LIN {X 0,Y 75.955,Z 312.798,A -85,B 0,C 180,E1 -27969.999,E2 -27969.999} C_VEL
LIN {X 0,Y 72.056,Z 313.683,A -85,B 0,C 180,E1 -27975.335,E2 -27975.335} C_VEL
LIN {X 0,Y 70.252,Z 314.024,A -85,B 0,C 180,E1 -27979.881,E2 -27979.881} C_VEL
LIN {X 0,Y 69.991,Z 314.033,A -85,B 0,C 180,E1 -27981.483,E2 -27981.483} C_VEL
LIN {X 0,Y 69.758,Z 313.788,A -85,B 0,C 180,E1 -27989.996,E2 -27989.996} C_VEL
LIN {X 0,Y 70.22,Z 313.122,A -85,B 0,C 180,E1 -27995.74,E2 -27995.74} C_VEL
LIN {X 0,Y 71.125,Z 312.075,A -85,B 0,C 180,E1 -28001.393,E2 -28001.393} C_VEL
LIN {X 0,Y 72.573,Z 310.585,A -85,B 0,C 180,E1 -28006.884,E2 -28006.884} C_VEL
LIN {X 0,Y 75.758,Z 307.579,A -85,B 0,C 180,E1 -28014.668,E2 -28014.668} C_VEL
LIN {X 0,Y 80.142,Z 303.529,A -85,B 0,C 180,E1 -28021.74,E2 -28021.74} C_VEL
LIN {X 0,Y 86.545,Z 297.313,A -85,B 0,C 180,E1 -28028.995,E2 -28028.995} C_VEL
LIN {X 0,Y 92.996,Z 290.542,A -85,B 0,C 180,E1 -28034.343,E2 -28034.343} C_VEL
LIN {X 0,Y 98.789,Z 283.636,A -85,B 0,C 180,E1 -28038.321,E2 -28038.321} C_VEL
LIN {X 0,Y 101.219,Z 280.484,A -85,B 0,C 180,E1 -28039.788,E2 -28039.788} C_VEL
LIN {X 0,Y 102.858,Z 276.343,A -85,B 0,C 180,E1 -28042.553,E2 -28042.553} C_VEL
LIN {X 0,Y 103.486,Z 273.641,A -85,B 0,C 180,E1 -28044.572,E2 -28044.572} C_VEL
LIN {X 0,Y 103.73,Z 270.638,A -85,B 0,C 180,E1 -28047.177,E2 -28047.177} C_VEL
LIN {X 0,Y 103.119,Z 265.886,A -85,B 0,C 180,E1 -28052.362,E2 -28052.362} C_VEL
LIN {X 0,Y 102.624,Z 263.228,A -85,B 0,C 180,E1 -28055.738,E2 -28055.738} C_VEL
LIN {X 0,Y 101.676,Z 259.362,A -85,B 0,C 180,E1 -28061.877,E2 -28061.877} C_VEL
LIN {X 0,Y 100.935,Z 256.73,A -85,B 0,C 180,E1 -28067.942,E2 -28067.942} C_VEL
LIN {X 0,Y 100.648,Z 254.765,A -85,B 0,C 180,E1 -28075.995,E2 -28075.995} C_VEL
LIN {X 0,Y 100.96,Z 254.248,A -85,B 0,C 180,E1 -28079.999,E2 -28079.999} C_VEL
LIN {X 0,Y 101.079,Z 256.427,A -85,B 0,C 180,E1 -28087.993,E2 -28087.993} C_VEL
LIN {X 0,Y 101.672,Z 257.847,A -85,B 0,C 180,E1 -28091.968,E2 -28091.968} C_VEL
LIN {X 0,Y 102.317,Z 259.954,A -85,B 0,C 180,E1 -28095.946,E2 -28095.946} C_VEL
LIN {X 0,Y 102.785,Z 262.952,A -85,B 0,C 180,E1 -28099.991,E2 -28099.991} C_VEL
LIN {X 0,Y 103.035,Z 267.977,A -85,B 0,C 180,E1 -28105.157,E2 -28105.157} C_VEL
LIN {X 0,Y 103.023,Z 272.964,A -85,B 0,C 180,E1 -28109.641,E2 -28109.641} C_VEL
LIN {X 0,Y 102.775,Z 275.854,A -85,B 0,C 180,E1 -28112.002,E2 -28112.002} C_VEL
LIN {X 0,Y 100.768,Z 280.852,A -85,B 0,C 180,E1 -28114.976,E2 -28114.976} C_VEL
LIN {X 0,Y 97.27,Z 287.517,A -85,B 0,C 180,E1 -28119.049,E2 -28119.049} C_VEL
LIN {X 0,Y 90.366,Z 295.686,A -85,B 0,C 180,E1 -28124.004,E2 -28124.004} C_VEL
LIN {X 0,Y 85.188,Z 301.246,A -85,B 0,C 180,E1 -28128.708,E2 -28128.708} C_VEL
LIN {X 0,Y 79.619,Z 306.676,A -85,B 0,C 180,E1 -28134.994,E2 -28134.994} C_VEL
LIN {X 0,Y 75.07,Z 310.919,A -85,B 0,C 180,E1 -28142.096,E2 -28142.096} C_VEL
LIN {X 0,Y 72.862,Z 313.178,A -85,B 0,C 180,E1 -28147.311,E2 -28147.311} C_VEL
LIN {X 0,Y 71.207,Z 314.96,A -85,B 0,C 180,E1 -28152.782,E2 -28152.782} C_VEL
LIN {X 0,Y 70.138,Z 316.312,A -85,B 0,C 180,E1 -28158.444,E2 -28158.444} C_VEL
LIN {X 0,Y 69.618,Z 317.268,A -85,B 0,C 180,E1 -28164.21,E2 -28164.21} C_VEL
LIN {X 0,Y 69.673,Z 317.834,A -85,B 0,C 180,E1 -28170.004,E2 -28170.004} C_VEL
LIN {X 0,Y 69.621,Z 317.95,A -85,B 0,C 180,E1 -28175.797,E2 -28175.797} C_VEL
LIN {X 0,Y 70.144,Z 317.665,A -85,B 0,C 180,E1 -28181.563,E2 -28181.563} C_VEL
LIN {X 0,Y 72.933,Z 315.942,A -85,B 0,C 180,E1 -28192.674,E2 -28192.674} C_VEL
LIN {X 0,Y 75.178,Z 314.45,A -85,B 0,C 180,E1 -28197.869,E2 -28197.869} C_VEL
LIN {X 0,Y 79.764,Z 311.427,A -85,B 0,C 180,E1 -28204.941,E2 -28204.941} C_VEL
LIN {X 0,Y 85.398,Z 307.36,A -85,B 0,C 180,E1 -28211.177,E2 -28211.177} C_VEL
LIN {X 0,Y 92.891,Z 301.121,A -85,B 0,C 180,E1 -28217.532,E2 -28217.532} C_VEL
LIN {X 0,Y 100.186,Z 294.343,A -85,B 0,C 180,E1 -28222.108,E2 -28222.108} C_VEL
LIN {X 0,Y 102.526,Z 291.722,A -85,B 0,C 180,E1 -28223.652,E2 -28223.652} C_VEL
LIN {X 0,Y 106.564,Z 285.03,A -85,B 0,C 180,E1 -28228.157,E2 -28228.157} C_VEL
LIN {X 0,Y 107.391,Z 281.213,A -85,B 0,C 180,E1 -28231.636,E2 -28231.636} C_VEL
LIN {X 0,Y 107.939,Z 276.036,A -85,B 0,C 180,E1 -28237.005,E2 -28237.005} C_VEL
LIN {X 0,Y 108.074,Z 272.768,A -85,B 0,C 180,E1 -28241.026,E2 -28241.026} C_VEL
LIN {X 0,Y 108.135,Z 270.019,A -85,B 0,C 180,E1 -28244.932,E2 -28244.932} C_VEL
LIN {X 0,Y 108.02,Z 268.068,A -85,B 0,C 180,E1 -28248.745,E2 -28248.745} C_VEL
LIN {X 0,Y 107.866,Z 266.689,A -85,B 0,C 180,E1 -28252.513,E2 -28252.513} C_VEL
LIN {X 0,Y 107.979,Z 265.237,A -85,B 0,C 180,E1 -28260.001,E2 -28260.001} C_VEL
LIN {X 0,Y 107.676,Z 266.885,A -85,B 0,C 180,E1 -28267.765,E2 -28267.765} C_VEL
LIN {X 0,Y 107.883,Z 268.439,A -85,B 0,C 180,E1 -28272.273,E2 -28272.273} C_VEL
LIN {X 0,Y 108.215,Z 270.725,A -85,B 0,C 180,E1 -28276.994,E2 -28276.994} C_VEL
LIN {X 0,Y 108.545,Z 274.554,A -85,B 0,C 180,E1 -28282.861,E2 -28282.861} C_VEL
LIN {X 0,Y 108.197,Z 278.26,A -85,B 0,C 180,E1 -28287.046,E2 -28287.046} C_VEL
LIN {X 0,Y 107.345,Z 282.888,A -85,B 0,C 180,E1 -28291.667,E2 -28291.667} C_VEL
LIN {X 0,Y 106.008,Z 285.83,A -85,B 0,C 180,E1 -28294.035,E2 -28294.035} C_VEL
LIN {X 0,Y 104.982,Z 287.233,A -85,B 0,C 180,E1 -28294.909,E2 -28294.909} C_VEL
LIN {X 0,Y 97.412,Z 294.692,A -85,B 0,C 180,E1 -28299.143,E2 -28299.143} C_VEL
LIN {X 0,Y 89.39,Z 301.569,A -85,B 0,C 180,E1 -28304.96,E2 -28304.96} C_VEL
LIN {X 0,Y 83.435,Z 306.095,A -85,B 0,C 180,E1 -28310.82,E2 -28310.82} C_VEL
LIN {X 0,Y 77.622,Z 309.911,A -85,B 0,C 180,E1 -28318.44,E2 -28318.44} C_VEL
LIN {X 0,Y 73.212,Z 312.551,A -85,B 0,C 180,E1 -28327.417,E2 -28327.417} C_VEL
LIN {X 0,Y 71.531,Z 313.461,A -85,B 0,C 180,E1 -28332.855,E2 -28332.855} C_VEL
LIN {X 0,Y 69.991,Z 314.033,A -85,B 0,C 180,E1 -28341.483,E2 -28341.483} C_VEL
LIN {X 0,Y 69.438,Z 314.073,A -85,B 0,C 180,E1 -28344.684,E2 -28344.684} C_VEL
LIN {X 0,Y 68.018,Z 313.906,A -85,B 0,C 180,E1 -28349.481,E2 -28349.481} C_VEL
LIN {X 0,Y 64.974,Z 312.491,A -85,B 0,C 180,E1 -28361.198,E2 -28361.198} C_VEL
LIN {X 0,Y 65.187,Z 311.42,A -85,B 0,C 180,E1 -28366.375,E2 -28366.375} C_VEL
LIN {X 0,Y 65.618,Z 310.972,A -85,B 0,C 180,E1 -28368.043,E2 -28368.043} C_VEL
LIN {X 0,Y 69.372,Z 307.82,A -85,B 0,C 180,E1 -28377.116,E2 -28377.116} C_VEL
LIN {X 0,Y 74.216,Z 303.782,A -85,B 0,C 180,E1 -28384.616,E2 -28384.616} C_VEL
LIN {X 0,Y 81.161,Z 297.581,A -85,B 0,C 180,E1 -28392.143,E2 -28392.143} C_VEL
LIN {X 0,Y 88.063,Z 290.826,A -85,B 0,C 180,E1 -28397.57,E2 -28397.57} C_VEL
LIN {X 0,Y 95.523,Z 282.413,A -85,B 0,C 180,E1 -28402.262,E2 -28402.262} C_VEL
LIN {X 0,Y 96.961,Z 279.827,A -85,B 0,C 180,E1 -28403.959,E2 -28403.959} C_VEL
LIN {X 0,Y 97.919,Z 277.001,A -85,B 0,C 180,E1 -28406.203,E2 -28406.203} C_VEL
LIN {X 0,Y 98.319,Z 274.084,A -85,B 0,C 180,E1 -28409.056,E2 -28409.056} C_VEL
LIN {X 0,Y 98.185,Z 271.419,A -85,B 0,C 180,E1 -28412.301,E2 -28412.301} C_VEL
LIN {X 0,Y 97.853,Z 268.184,A -85,B 0,C 180,E1 -28416.731,E2 -28416.731} C_VEL
LIN {X 0,Y 97.258,Z 264.548,A -85,B 0,C 180,E1 -28423.198,E2 -28423.198} C_VEL
LIN {X 0,Y 96.959,Z 262.844,A -85,B 0,C 180,E1 -28427.439,E2 -28427.439} C_VEL
LIN {X 0,Y 96.783,Z 260.823,A -85,B 0,C 180,E1 -28435.835,E2 -28435.835} C_VEL
LIN {X 0,Y 97.132,Z 260.307,A -85,B 0,C 180,E1 -28439.999,E2 -28439.999} C_VEL
LIN {X 0,Y 97.154,Z 262.517,A -85,B 0,C 180,E1 -28448.318,E2 -28448.318} C_VEL
LIN {X 0,Y 97.649,Z 264.033,A -85,B 0,C 180,E1 -28452.468,E2 -28452.468} C_VEL
LIN {X 0,Y 97.966,Z 266.405,A -85,B 0,C 180,E1 -28456.675,E2 -28456.675} C_VEL
LIN {X 0,Y 98.12,Z 267.867,A -85,B 0,C 180,E1 -28458.802,E2 -28458.802} C_VEL
LIN {X 0,Y 97.911,Z 272.888,A -85,B 0,C 180,E1 -28464.374,E2 -28464.374} C_VEL
LIN {X 0,Y 97.466,Z 277.636,A -85,B 0,C 180,E1 -28468.998,E2 -28468.998} C_VEL
LIN {X 0,Y 96.932,Z 279.503,A -85,B 0,C 180,E1 -28470.499,E2 -28470.499} C_VEL
LIN {X 0,Y 93.687,Z 285.648,A -85,B 0,C 180,E1 -28474.405,E2 -28474.405} C_VEL
LIN {X 0,Y 91.691,Z 288.714,A -85,B 0,C 180,E1 -28476.418,E2 -28476.418} C_VEL
LIN {X 0,Y 84.392,Z 296.628,A -85,B 0,C 180,E1 -28481.462,E2 -28481.462} C_VEL
LIN {X 0,Y 77.841,Z 302.947,A -85,B 0,C 180,E1 -28487.387,E2 -28487.387} C_VEL
LIN {X 0,Y 72.098,Z 307.974,A -85,B 0,C 180,E1 -28494.214,E2 -28494.214} C_VEL
LIN {X 0,Y 67.496,Z 311.866,A -85,B 0,C 180,E1 -28502.066,E2 -28502.066} C_VEL
LIN {X 0,Y 64.441,Z 314.737,A -85,B 0,C 180,E1 -28510.908,E2 -28510.908} C_VEL
LIN {X 0,Y 63.173,Z 316.095,A -85,B 0,C 180,E1 -28517.149,E2 -28517.149} C_VEL
LIN {X 0,Y 62.553,Z 317.057,A -85,B 0,C 180,E1 -28523.554,E2 -28523.554} C_VEL
LIN {X 0,Y 62.564,Z 317.628,A -85,B 0,C 180,E1 -28530.004,E2 -28530.004} C_VEL
LIN {X 0,Y 62.556,Z 317.754,A -85,B 0,C 180,E1 -28536.455,E2 -28536.455} C_VEL
LIN {X 0,Y 64.469,Z 316.812,A -85,B 0,C 180,E1 -28549.092,E2 -28549.092} C_VEL
LIN {X 0,Y 66.394,Z 315.762,A -85,B 0,C 180,E1 -28555.053,E2 -28555.053} C_VEL
LIN {X 0,Y 68.957,Z 314.281,A -85,B 0,C 180,E1 -28560.639,E2 -28560.639} C_VEL
LIN {X 0,Y 74.036,Z 311.27,A -85,B 0,C 180,E1 -28568.101,E2 -28568.101} C_VEL
LIN {X 0,Y 80.179,Z 307.215,A -85,B 0,C 180,E1 -28574.526,E2 -28574.526} C_VEL
LIN {X 0,Y 88.233,Z 300.99,A -85,B 0,C 180,E1 -28580.951,E2 -28580.951} C_VEL
LIN {X 0,Y 95.975,Z 294.228,A -85,B 0,C 180,E1 -28585.467,E2 -28585.467} C_VEL
LIN {X 0,Y 97.202,Z 292.973,A -85,B 0,C 180,E1 -28586.251,E2 -28586.251} C_VEL
LIN {X 0,Y 100.572,Z 288.15,A -85,B 0,C 180,E1 -28589.722,E2 -28589.722} C_VEL
LIN {X 0,Y 101.23,Z 286.76,A -85,B 0,C 180,E1 -28590.924,E2 -28590.924} C_VEL
LIN {X 0,Y 102.278,Z 282.398,A -85,B 0,C 180,E1 -28595.652,E2 -28595.652} C_VEL
LIN {X 0,Y 102.847,Z 278.852,A -85,B 0,C 180,E1 -28600.022,E2 -28600.022} C_VEL
LIN {X 0,Y 103.165,Z 276.019,A -85,B 0,C 180,E1 -28604.188,E2 -28604.188} C_VEL
LIN {X 0,Y 103.363,Z 273.814,A -85,B 0,C 180,E1 -28608.231,E2 -28608.231} C_VEL
LIN {X 0,Y 103.361,Z 272.372,A -85,B 0,C 180,E1 -28612.185,E2 -28612.185} C_VEL
LIN {X 0,Y 103.556,Z 270.864,A -85,B 0,C 180,E1 -28620.001,E2 -28620.001} C_VEL
LIN {X 0,Y 103.125,Z 272.419,A -85,B 0,C 180,E1 -28627.835,E2 -28627.835} C_VEL
LIN {X 0,Y 103.164,Z 273.663,A -85,B 0,C 180,E1 -28631.794,E2 -28631.794} C_VEL
LIN {X 0,Y 103.269,Z 276.393,A -85,B 0,C 180,E1 -28637.683,E2 -28637.683} C_VEL
LIN {X 0,Y 103.251,Z 279.001,A -85,B 0,C 180,E1 -28641.986,E2 -28641.986} C_VEL
LIN {X 0,Y 102.452,Z 283.012,A -85,B 0,C 180,E1 -28646.905,E2 -28646.905} C_VEL
LIN {X 0,Y 101.988,Z 284.706,A -85,B 0,C 180,E1 -28648.842,E2 -28648.842} C_VEL
LIN {X 0,Y 100.629,Z 287.643,A -85,B 0,C 180,E1 -28651.611,E2 -28651.611} C_VEL
LIN {X 0,Y 95.729,Z 292.503,A -85,B 0,C 180,E1 -28654.319,E2 -28654.319} C_VEL
LIN {X 0,Y 89.284,Z 297.98,A -85,B 0,C 180,E1 -28658.08,E2 -28658.08} C_VEL
LIN {X 0,Y 82.425,Z 303.193,A -85,B 0,C 180,E1 -28663.262,E2 -28663.262} C_VEL
LIN {X 0,Y 76.073,Z 307.488,A -85,B 0,C 180,E1 -28669.706,E2 -28669.706} C_VEL
LIN {X 0,Y 72.408,Z 309.696,A -85,B 0,C 180,E1 -28674.381,E2 -28674.381} C_VEL
LIN {X 0,Y 69.213,Z 311.423,A -85,B 0,C 180,E1 -28679.487,E2 -28679.487} C_VEL
LIN {X 0,Y 64.762,Z 313.646,A -85,B 0,C 180,E1 -28690.997,E2 -28690.997} C_VEL
LIN {X 0,Y 62.938,Z 314.236,A -85,B 0,C 180,E1 -28700.978,E2 -28700.978} C_VEL
LIN {X 0,Y 62.679,Z 313.994,A -85,B 0,C 180,E1 -28709.996,E2 -28709.996} C_VEL
LIN {X 0,Y 63.18,Z 313.334,A -85,B 0,C 180,E1 -28716.382,E2 -28716.382} C_VEL
LIN {X 0,Y 64.189,Z 312.294,A -85,B 0,C 180,E1 -28722.644,E2 -28722.644} C_VEL
LIN {X 0,Y 65.618,Z 310.972,A -85,B 0,C 180,E1 -28728.043,E2 -28728.043} C_VEL
LIN {X 0,Y 66.735,Z 309.623,A -85,B 0,C 180,E1 -28732.928,E2 -28732.928} C_VEL
LIN {X 0,Y 67.72,Z 306.86,A -85,B 0,C 180,E1 -28741.014,E2 -28741.014} C_VEL
LIN {X 0,Y 69.774,Z 303.403,A -85,B 0,C 180,E1 -28748.598,E2 -28748.598} C_VEL
LIN {X 0,Y 72.402,Z 300.889,A -85,B 0,C 180,E1 -28752.383,E2 -28752.383} C_VEL
LIN {X 0,Y 79.684,Z 294.661,A -85,B 0,C 180,E1 -28758.553,E2 -28758.553} C_VEL
LIN {X 0,Y 87.32,Z 287.157,A -85,B 0,C 180,E1 -28763.585,E2 -28763.585} C_VEL
LIN {X 0,Y 90.886,Z 283.208,A -85,B 0,C 180,E1 -28765.616,E2 -28765.616} C_VEL
LIN {X 0,Y 91.978,Z 281.164,A -85,B 0,C 180,E1 -28767.182,E2 -28767.182} C_VEL
LIN {X 0,Y 92.61,Z 279.392,A -85,B 0,C 180,E1 -28768.899,E2 -28768.899} C_VEL
LIN {X 0,Y 92.87,Z 277.921,A -85,B 0,C 180,E1 -28770.534,E2 -28770.534} C_VEL
LIN {X 0,Y 92.877,Z 274.63,A -85,B 0,C 180,E1 -28775.22,E2 -28775.22} C_VEL
LIN {X 0,Y 92.789,Z 271.95,A -85,B 0,C 180,E1 -28779.698,E2 -28779.698} C_VEL
LIN {X 0,Y 92.742,Z 270.542,A -85,B 0,C 180,E1 -28782.354,E2 -28782.354} C_VEL
LIN {X 0,Y 92.552,Z 268.768,A -85,B 0,C 180,E1 -28786.831,E2 -28786.831} C_VEL
LIN {X 0,Y 92.461,Z 267.552,A -85,B 0,C 180,E1 -28791.255,E2 -28791.255} C_VEL
LIN {X 0,Y 92.585,Z 266.672,A -85,B 0,C 180,E1 -28795.646,E2 -28795.646} C_VEL
LIN {X 0,Y 92.963,Z 266.166,A -85,B 0,C 180,E1 -28799.999,E2 -28799.999} C_VEL
LIN {X 0,Y 93.061,Z 269.154,A -85,B 0,C 180,E1 -28810.995,E2 -28810.995} C_VEL
LIN {X 0,Y 93.254,Z 271.189,A -85,B 0,C 180,E1 -28815.293,E2 -28815.293} C_VEL
LIN {X 0,Y 93.259,Z 272.612,A -85,B 0,C 180,E1 -28817.543,E2 -28817.543} C_VEL
LIN {X 0,Y 92.739,Z 276.431,A -85,B 0,C 180,E1 -28822.266,E2 -28822.266} C_VEL
LIN {X 0,Y 91.913,Z 281.062,A -85,B 0,C 180,E1 -28827.308,E2 -28827.308} C_VEL
LIN {X 0,Y 90.911,Z 283.114,A -85,B 0,C 180,E1 -28828.871,E2 -28828.871} C_VEL
LIN {X 0,Y 87.528,Z 288.405,A -85,B 0,C 180,E1 -28832.545,E2 -28832.545} C_VEL
LIN {X 0,Y 82.366,Z 293.881,A -85,B 0,C 180,E1 -28835.857,E2 -28835.857} C_VEL
LIN {X 0,Y 75.004,Z 300.708,A -85,B 0,C 180,E1 -28841.453,E2 -28841.453} C_VEL
LIN {X 0,Y 68.403,Z 306.168,A -85,B 0,C 180,E1 -28848.109,E2 -28848.109} C_VEL
LIN {X 0,Y 62.842,Z 310.439,A -85,B 0,C 180,E1 -28856.009,E2 -28856.009} C_VEL
LIN {X 0,Y 59.914,Z 312.707,A -85,B 0,C 180,E1 -28862.024,E2 -28862.024} C_VEL
LIN {X 0,Y 57.732,Z 314.513,A -85,B 0,C 180,E1 -28868.587,E2 -28868.587} C_VEL
LIN {X 0,Y 56.261,Z 315.878,A -85,B 0,C 180,E1 -28875.538,E2 -28875.538} C_VEL
LIN {X 0,Y 55.511,Z 316.846,A -85,B 0,C 180,E1 -28882.732,E2 -28882.732} C_VEL
LIN {X 0,Y 55.475,Z 317.423,A -85,B 0,C 180,E1 -28890.005,E2 -28890.005} C_VEL
LIN {X 0,Y 55.514,Z 317.56,A -85,B 0,C 180,E1 -28897.278,E2 -28897.278} C_VEL
LIN {X 0,Y 57.779,Z 316.627,A -85,B 0,C 180,E1 -28911.405,E2 -28911.405} C_VEL
LIN {X 0,Y 59.996,Z 315.582,A -85,B 0,C 180,E1 -28917.944,E2 -28917.944} C_VEL
LIN {X 0,Y 62.934,Z 314.113,A -85,B 0,C 180,E1 -28923.945,E2 -28923.945} C_VEL
LIN {X 0,Y 68.56,Z 311.112,A -85,B 0,C 180,E1 -28931.784,E2 -28931.784} C_VEL
LIN {X 0,Y 76.758,Z 306.048,A -85,B 0,C 180,E1 -28939.59,E2 -28939.59} C_VEL
LIN {X 0,Y 85.25,Z 299.849,A -85,B 0,C 180,E1 -28945.527,E2 -28945.527} C_VEL
LIN {X 0,Y 92.072,Z 294.113,A -85,B 0,C 180,E1 -28949.173,E2 -28949.173} C_VEL
LIN {X 0,Y 95.249,Z 290.122,A -85,B 0,C 180,E1 -28952.302,E2 -28952.302} C_VEL
LIN {X 0,Y 96.261,Z 287.575,A -85,B 0,C 180,E1 -28955.178,E2 -28955.178} C_VEL
LIN {X 0,Y 97.295,Z 283.977,A -85,B 0,C 180,E1 -28959.888,E2 -28959.888} C_VEL
LIN {X 0,Y 98.086,Z 280.469,A -85,B 0,C 180,E1 -28965.477,E2 -28965.477} C_VEL
LIN {X 0,Y 98.338,Z 279.317,A -85,B 0,C 180,E1 -28967.62,E2 -28967.62} C_VEL
LIN {X 0,Y 98.478,Z 277.804,A -85,B 0,C 180,E1 -28971.795,E2 -28971.795} C_VEL
LIN {X 0,Y 98.61,Z 276.782,A -85,B 0,C 180,E1 -28976.167,E2 -28976.167} C_VEL
LIN {X 0,Y 98.836,Z 276.237,A -85,B 0,C 180,E1 -28980.001,E2 -28980.001} C_VEL
LIN {X 0,Y 98.214,Z 277.777,A -85,B 0,C 180,E1 -28988.229,E2 -28988.229} C_VEL
LIN {X 0,Y 98.119,Z 279.1,A -85,B 0,C 180,E1 -28992.41,E2 -28992.41} C_VEL
LIN {X 0,Y 98.04,Z 280.861,A -85,B 0,C 180,E1 -28996.664,E2 -28996.664} C_VEL
LIN {X 0,Y 97.763,Z 283.271,A -85,B 0,C 180,E1 -29001.067,E2 -29001.067} C_VEL
LIN {X 0,Y 96.663,Z 286.791,A -85,B 0,C 180,E1 -29005.865,E2 -29005.865} C_VEL
LIN {X 0,Y 95.743,Z 288.803,A -85,B 0,C 180,E1 -29008.256,E2 -29008.256} C_VEL
LIN {X 0,Y 94.676,Z 290.141,A -85,B 0,C 180,E1 -29009.283,E2 -29009.283} C_VEL
LIN {X 0,Y 86.405,Z 297.105,A -85,B 0,C 180,E1 -29013.518,E2 -29013.518} C_VEL
LIN {X 0,Y 78.409,Z 302.867,A -85,B 0,C 180,E1 -29018.863,E2 -29018.863} C_VEL
LIN {X 0,Y 70.778,Z 307.643,A -85,B 0,C 180,E1 -29025.965,E2 -29025.965} C_VEL
LIN {X 0,Y 66.758,Z 309.858,A -85,B 0,C 180,E1 -29030.826,E2 -29030.826} C_VEL
LIN {X 0,Y 63.172,Z 311.596,A -85,B 0,C 180,E1 -29036.2,E2 -29036.2} C_VEL
LIN {X 0,Y 58.085,Z 313.83,A -85,B 0,C 180,E1 -29048.713,E2 -29048.713} C_VEL
LIN {X 0,Y 56.522,Z 314.367,A -85,B 0,C 180,E1 -29055.596,E2 -29055.596} C_VEL
LIN {X 0,Y 55.692,Z 314.479,A -85,B 0,C 180,E1 -29062.746,E2 -29062.746} C_VEL
LIN {X 0,Y 55.591,Z 314.2,A -85,B 0,C 180,E1 -29069.995,E2 -29069.995} C_VEL
LIN {X 0,Y 56.136,Z 313.545,A -85,B 0,C 180,E1 -29077.187,E2 -29077.187} C_VEL
LIN {X 0,Y 57.283,Z 312.513,A -85,B 0,C 180,E1 -29084.198,E2 -29084.198} C_VEL
LIN {X 0,Y 59.154,Z 311.042,A -85,B 0,C 180,E1 -29090.874,E2 -29090.874} C_VEL
LIN {X 0,Y 63.146,Z 308.061,A -85,B 0,C 180,E1 -29100.048,E2 -29100.048} C_VEL
LIN {X 0,Y 68.486,Z 304.037,A -85,B 0,C 180,E1 -29107.996,E2 -29107.996} C_VEL
LIN {X 0,Y 72.402,Z 300.889,A -85,B 0,C 180,E1 -29112.383,E2 -29112.383} C_VEL
LIN {X 0,Y 76.26,Z 297.24,A -85,B 0,C 180,E1 -29116.848,E2 -29116.848} C_VEL
LIN {X 0,Y 79.485,Z 293.298,A -85,B 0,C 180,E1 -29121.286,E2 -29121.286} C_VEL
LIN {X 0,Y 82.645,Z 289.036,A -85,B 0,C 180,E1 -29125.484,E2 -29125.484} C_VEL
LIN {X 0,Y 86.2,Z 284.363,A -85,B 0,C 180,E1 -29129.147,E2 -29129.147} C_VEL
LIN {X 0,Y 87.106,Z 282.499,A -85,B 0,C 180,E1 -29131.045,E2 -29131.045} C_VEL
LIN {X 0,Y 87.439,Z 280.718,A -85,B 0,C 180,E1 -29133.564,E2 -29133.564} C_VEL
LIN {X 0,Y 87.75,Z 277.549,A -85,B 0,C 180,E1 -29138.873,E2 -29138.873} C_VEL
LIN {X 0,Y 87.814,Z 275.307,A -85,B 0,C 180,E1 -29143.796,E2 -29143.796} C_VEL
LIN {X 0,Y 87.824,Z 273.171,A -85,B 0,C 180,E1 -29150.789,E2 -29150.789} C_VEL
LIN {X 0,Y 88.071,Z 272.274,A -85,B 0,C 180,E1 -29155.422,E2 -29155.422} C_VEL
LIN {X 0,Y 88.49,Z 271.776,A -85,B 0,C 180,E1 -29159.999,E2 -29159.999} C_VEL
LIN {X 0,Y 88.259,Z 273.997,A -85,B 0,C 180,E1 -29169.163,E2 -29169.163} C_VEL
LIN {X 0,Y 88.35,Z 275.805,A -85,B 0,C 180,E1 -29173.805,E2 -29173.805} C_VEL
LIN {X 0,Y 87.833,Z 278.866,A -85,B 0,C 180,E1 -29178.666,E2 -29178.666} C_VEL
LIN {X 0,Y 86.745,Z 283.013,A -85,B 0,C 180,E1 -29183.896,E2 -29183.896} C_VEL
LIN {X 0,Y 85.9,Z 284.975,A -85,B 0,C 180,E1 -29185.86,E2 -29185.86} C_VEL
LIN {X 0,Y 82.522,Z 289.579,A -85,B 0,C 180,E1 -29189.212,E2 -29189.212} C_VEL
LIN {X 0,Y 74.455,Z 297.113,A -85,B 0,C 180,E1 -29194.136,E2 -29194.136} C_VEL
LIN {X 0,Y 65.596,Z 304.247,A -85,B 0,C 180,E1 -29201.422,E2 -29201.422} C_VEL
LIN {X 0,Y 59.015,Z 308.914,A -85,B 0,C 180,E1 -29209.091,E2 -29209.091} C_VEL
LIN {X 0,Y 53.706,Z 312.471,A -85,B 0,C 180,E1 -29218.445,E2 -29218.445} C_VEL
LIN {X 0,Y 51.145,Z 314.289,A -85,B 0,C 180,E1 -29225.662,E2 -29225.662} C_VEL
LIN {X 0,Y 49.382,Z 315.66,A -85,B 0,C 180,E1 -29233.47,E2 -29233.47} C_VEL
LIN {X 0,Y 48.471,Z 316.634,A -85,B 0,C 180,E1 -29241.669,E2 -29241.669} C_VEL
LIN {X 0,Y 48.372,Z 317.217,A -85,B 0,C 180,E1 -29250.006,E2 -29250.006} C_VEL
LIN {X 0,Y 48.474,Z 317.364,A -85,B 0,C 180,E1 -29258.341,E2 -29258.341} C_VEL
LIN {X 0,Y 51.195,Z 316.441,A -85,B 0,C 180,E1 -29274.324,E2 -29274.324} C_VEL
LIN {X 0,Y 53.789,Z 315.402,A -85,B 0,C 180,E1 -29281.513,E2 -29281.513} C_VEL
LIN {X 0,Y 57.168,Z 313.946,A -85,B 0,C 180,E1 -29287.931,E2 -29287.931} C_VEL
LIN {X 0,Y 63.409,Z 310.954,A -85,B 0,C 180,E1 -29296.092,E2 -29296.092} C_VEL
LIN {X 0,Y 70.716,Z 306.923,A -85,B 0,C 180,E1 -29302.663,E2 -29302.663} C_VEL
LIN {X 0,Y 80.015,Z 300.73,A -85,B 0,C 180,E1 -29308.912,E2 -29308.912} C_VEL
LIN {X 0,Y 87.183,Z 295.234,A -85,B 0,C 180,E1 -29312.464,E2 -29312.464} C_VEL
LIN {X 0,Y 89.542,Z 292.736,A -85,B 0,C 180,E1 -29314.502,E2 -29314.502} C_VEL
LIN {X 0,Y 90.652,Z 290.58,A -85,B 0,C 180,E1 -29317.194,E2 -29317.194} C_VEL
LIN {X 0,Y 91.984,Z 287.226,A -85,B 0,C 180,E1 -29322.206,E2 -29322.206} C_VEL
LIN {X 0,Y 92.843,Z 284.701,A -85,B 0,C 180,E1 -29326.875,E2 -29326.875} C_VEL
LIN {X 0,Y 93.118,Z 283.788,A -85,B 0,C 180,E1 -29328.855,E2 -29328.855} C_VEL
LIN {X 0,Y 93.256,Z 282.972,A -85,B 0,C 180,E1 -29331.332,E2 -29331.332} C_VEL
LIN {X 0,Y 93.512,Z 281.908,A -85,B 0,C 180,E1 -29335.691,E2 -29335.691} C_VEL
LIN {X 0,Y 93.805,Z 281.306,A -85,B 0,C 180,E1 -29340.001,E2 -29340.001} C_VEL
LIN {X 0,Y 93,Z 282.694,A -85,B 0,C 180,E1 -29347.781,E2 -29347.781} C_VEL
LIN {X 0,Y 92.747,Z 284.25,A -85,B 0,C 180,E1 -29353.141,E2 -29353.141} C_VEL
LIN {X 0,Y 92.41,Z 286.092,A -85,B 0,C 180,E1 -29357.712,E2 -29357.712} C_VEL
LIN {X 0,Y 91.953,Z 287.681,A -85,B 0,C 180,E1 -29360.67,E2 -29360.67} C_VEL
LIN {X 0,Y 91.02,Z 289.796,A -85,B 0,C 180,E1 -29363.913,E2 -29363.913} C_VEL
LIN {X 0,Y 89.925,Z 291.501,A -85,B 0,C 180,E1 -29366.005,E2 -29366.005} C_VEL
LIN {X 0,Y 81.277,Z 298.237,A -85,B 0,C 180,E1 -29370.153,E2 -29370.153} C_VEL
LIN {X 0,Y 73.656,Z 303.312,A -85,B 0,C 180,E1 -29374.926,E2 -29374.926} C_VEL
LIN {X 0,Y 65.821,Z 307.799,A -85,B 0,C 180,E1 -29381.631,E2 -29381.631} C_VEL
LIN {X 0,Y 61.389,Z 310.02,A -85,B 0,C 180,E1 -29386.613,E2 -29386.613} C_VEL
LIN {X 0,Y 57.384,Z 311.77,A -85,B 0,C 180,E1 -29392.237,E2 -29392.237} C_VEL
LIN {X 0,Y 51.503,Z 314.014,A -85,B 0,C 180,E1 -29405.831,E2 -29405.831} C_VEL
LIN {X 0,Y 49.671,Z 314.558,A -85,B 0,C 180,E1 -29413.557,E2 -29413.557} C_VEL
LIN {X 0,Y 48.648,Z 314.679,A -85,B 0,C 180,E1 -29421.689,E2 -29421.689} C_VEL
LIN {X 0,Y 48.492,Z 314.406,A -85,B 0,C 180,E1 -29429.994,E2 -29429.994} C_VEL
LIN {X 0,Y 49.127,Z 313.756,A -85,B 0,C 180,E1 -29438.219,E2 -29438.219} C_VEL
LIN {X 0,Y 50.447,Z 312.73,A -85,B 0,C 180,E1 -29446.172,E2 -29446.172} C_VEL
LIN {X 0,Y 52.578,Z 311.271,A -85,B 0,C 180,E1 -29453.634,E2 -29453.634} C_VEL
LIN {X 0,Y 57.129,Z 308.301,A -85,B 0,C 180,E1 -29463.605,E2 -29463.605} C_VEL
LIN {X 0,Y 63.044,Z 304.29,A -85,B 0,C 180,E1 -29471.97,E2 -29471.97} C_VEL
LIN {X 0,Y 71.299,Z 298.116,A -85,B 0,C 180,E1 -29479.801,E2 -29479.801} C_VEL
LIN {X 0,Y 79.192,Z 291.392,A -85,B 0,C 180,E1 -29485.163,E2 -29485.163} C_VEL
LIN {X 0,Y 85.705,Z 284.987,A -85,B 0,C 180,E1 -29488.722,E2 -29488.722} C_VEL
LIN {X 0,Y 86.2,Z 284.363,A -85,B 0,C 180,E1 -29489.147,E2 -29489.147} C_VEL
LIN {X 0,Y 87.266,Z 282.59,A -85,B 0,C 180,E1 -29490.781,E2 -29490.781} C_VEL
LIN {X 0,Y 87.507,Z 280.959,A -85,B 0,C 180,E1 -29493.33,E2 -29493.33} C_VEL
LIN {X 0,Y 86.651,Z 279.713,A -85,B 0,C 180,E1 -29497.106,E2 -29497.106} C_VEL
LIN {X 0,Y 83.938,Z 279.115,A -85,B 0,C 180,E1 -29504.281,E2 -29504.281} C_VEL
LIN {X 0,Y 82.865,Z 278.5,A -85,B 0,C 180,E1 -29510.426,E2 -29510.426} C_VEL
LIN {X 0,Y 83.193,Z 277.606,A -85,B 0,C 180,E1 -29515.153,E2 -29515.153} C_VEL
LIN {X 0,Y 83.685,Z 277.124,A -85,B 0,C 180,E1 -29519.999,E2 -29519.999} C_VEL
LIN {X 0,Y 83.308,Z 278.122,A -85,B 0,C 180,E1 -29524.838,E2 -29524.838} C_VEL
LIN {X 0,Y 83.241,Z 279.417,A -85,B 0,C 180,E1 -29529.72,E2 -29529.72} C_VEL
LIN {X 0,Y 83.209,Z 280.297,A -85,B 0,C 180,E1 -29532.189,E2 -29532.189} C_VEL
LIN {X 0,Y 82.649,Z 282.527,A -85,B 0,C 180,E1 -29536.415,E2 -29536.415} C_VEL
LIN {X 0,Y 81.229,Z 286.311,A -85,B 0,C 180,E1 -29541.803,E2 -29541.803} C_VEL
LIN {X 0,Y 80.299,Z 287.756,A -85,B 0,C 180,E1 -29543.239,E2 -29543.239} C_VEL
LIN {X 0,Y 77.823,Z 290.654,A -85,B 0,C 180,E1 -29545.451,E2 -29545.451} C_VEL
LIN {X 0,Y 68.894,Z 298.276,A -85,B 0,C 180,E1 -29550.473,E2 -29550.473} C_VEL
LIN {X 0,Y 61.12,Z 303.987,A -85,B 0,C 180,E1 -29556.412,E2 -29556.412} C_VEL
LIN {X 0,Y 53.83,Z 308.667,A -85,B 0,C 180,E1 -29564.115,E2 -29564.115} C_VEL
LIN {X 0,Y 47.768,Z 312.236,A -85,B 0,C 180,E1 -29573.958,E2 -29573.958} C_VEL
LIN {X 0,Y 44.738,Z 314.065,A -85,B 0,C 180,E1 -29581.892,E2 -29581.892} C_VEL
LIN {X 0,Y 42.599,Z 315.442,A -85,B 0,C 180,E1 -29590.742,E2 -29590.742} C_VEL
LIN {X 0,Y 41.444,Z 316.422,A -85,B 0,C 180,E1 -29600.244,E2 -29600.244} C_VEL
LIN {X 0,Y 41.285,Z 317.012,A -85,B 0,C 180,E1 -29610.007,E2 -29610.007} C_VEL
LIN {X 0,Y 41.448,Z 317.169,A -85,B 0,C 180,E1 -29619.768,E2 -29619.768} C_VEL
LIN {X 0,Y 44.788,Z 316.256,A -85,B 0,C 180,E1 -29638.088,E2 -29638.088} C_VEL
LIN {X 0,Y 47.847,Z 315.222,A -85,B 0,C 180,E1 -29645.987,E2 -29645.987} C_VEL
LIN {X 0,Y 51.743,Z 313.778,A -85,B 0,C 180,E1 -29652.778,E2 -29652.778} C_VEL
LIN {X 0,Y 58.682,Z 310.795,A -85,B 0,C 180,E1 -29661.122,E2 -29661.122} C_VEL
LIN {X 0,Y 66.623,Z 306.776,A -85,B 0,C 180,E1 -29667.556,E2 -29667.556} C_VEL
LIN {X 0,Y 76.585,Z 300.601,A -85,B 0,C 180,E1 -29673.474,E2 -29673.474} C_VEL
LIN {X 0,Y 82.606,Z 296.306,A -85,B 0,C 180,E1 -29676.147,E2 -29676.147} C_VEL
LIN {X 0,Y 83.924,Z 295.112,A -85,B 0,C 180,E1 -29677.096,E2 -29677.096} C_VEL
LIN {X 0,Y 84.67,Z 294.136,A -85,B 0,C 180,E1 -29678.296,E2 -29678.296} C_VEL
LIN {X 0,Y 86.307,Z 291.069,A -85,B 0,C 180,E1 -29683.442,E2 -29683.442} C_VEL
LIN {X 0,Y 86.93,Z 289.778,A -85,B 0,C 180,E1 -29685.964,E2 -29685.964} C_VEL
LIN {X 0,Y 87.756,Z 287.847,A -85,B 0,C 180,E1 -29690.784,E2 -29690.784} C_VEL
LIN {X 0,Y 88.12,Z 286.723,A -85,B 0,C 180,E1 -29695.427,E2 -29695.427} C_VEL
LIN {X 0,Y 88.482,Z 286.085,A -85,B 0,C 180,E1 -29700.001,E2 -29700.001} C_VEL
LIN {X 0,Y 87.557,Z 287.367,A -85,B 0,C 180,E1 -29707.65,E2 -29707.65} C_VEL
LIN {X 0,Y 87.496,Z 287.687,A -85,B 0,C 180,E1 -29709.246,E2 -29709.246} C_VEL
LIN {X 0,Y 86.741,Z 289.995,A -85,B 0,C 180,E1 -29716.473,E2 -29716.473} C_VEL
LIN {X 0,Y 85.717,Z 292.138,A -85,B 0,C 180,E1 -29720.828,E2 -29720.828} C_VEL
LIN {X 0,Y 83.994,Z 294.057,A -85,B 0,C 180,E1 -29723.017,E2 -29723.017} C_VEL
LIN {X 0,Y 74.998,Z 300.316,A -85,B 0,C 180,E1 -29727.098,E2 -29727.098} C_VEL
LIN {X 0,Y 66.573,Z 305.284,A -85,B 0,C 180,E1 -29732.376,E2 -29732.376} C_VEL
LIN {X 0,Y 58.828,Z 309.124,A -85,B 0,C 180,E1 -29739.053,E2 -29739.053} C_VEL
LIN {X 0,Y 51.931,Z 311.943,A -85,B 0,C 180,E1 -29747.413,E2 -29747.413} C_VEL
LIN {X 0,Y 45.1,Z 314.199,A -85,B 0,C 180,E1 -29762.124,E2 -29762.124} C_VEL
LIN {X 0,Y 42.888,Z 314.749,A -85,B 0,C 180,E1 -29770.863,E2 -29770.863} C_VEL
LIN {X 0,Y 41.641,Z 314.88,A -85,B 0,C 180,E1 -29780.277,E2 -29780.277} C_VEL
LIN {X 0,Y 41.41,Z 314.611,A -85,B 0,C 180,E1 -29789.993,E2 -29789.993} C_VEL
LIN {X 0,Y 42.128,Z 313.967,A -85,B 0,C 180,E1 -29799.596,E2 -29799.596} C_VEL
LIN {X 0,Y 43.674,Z 312.947,A -85,B 0,C 180,E1 -29808.766,E2 -29808.766} C_VEL
LIN {X 0,Y 46.166,Z 311.5,A -85,B 0,C 180,E1 -29817.165,E2 -29817.165} C_VEL
LIN {X 0,Y 51.367,Z 308.542,A -85,B 0,C 180,E1 -29827.992,E2 -29827.992} C_VEL
LIN {X 0,Y 57.967,Z 304.543,A -85,B 0,C 180,E1 -29836.662,E2 -29836.662} C_VEL
LIN {X 0,Y 66.948,Z 298.383,A -85,B 0,C 180,E1 -29844.434,E2 -29844.434} C_VEL
LIN {X 0,Y 75.369,Z 291.674,A -85,B 0,C 180,E1 -29849.588,E2 -29849.588} C_VEL
LIN {X 0,Y 81.203,Z 286.331,A -85,B 0,C 180,E1 -29852.469,E2 -29852.469} C_VEL
LIN {X 0,Y 81.837,Z 284.827,A -85,B 0,C 180,E1 -29854.57,E2 -29854.57} C_VEL
LIN {X 0,Y 82.447,Z 281.923,A -85,B 0,C 180,E1 -29860.063,E2 -29860.063} C_VEL
LIN {X 0,Y 82.744,Z 279.889,A -85,B 0,C 180,E1 -29865.236,E2 -29865.236} C_VEL
LIN {X 0,Y 82.865,Z 278.5,A -85,B 0,C 180,E1 -29870.426,E2 -29870.426} C_VEL
LIN {X 0,Y 82.439,Z 278.552,A -85,B 0,C 180,E1 -29873.114,E2 -29873.114} C_VEL
LIN {X 0,Y 81.018,Z 279.765,A -85,B 0,C 180,E1 -29876.595,E2 -29876.595} C_VEL
LIN {X 0,Y 78.387,Z 282.606,A -85,B 0,C 180,E1 -29882.918,E2 -29882.918} C_VEL
LIN {X 0,Y 78.126,Z 283.13,A -85,B 0,C 180,E1 -29884.879,E2 -29884.879} C_VEL
LIN {X 0,Y 77.93,Z 284.554,A -85,B 0,C 180,E1 -29890.39,E2 -29890.39} C_VEL
LIN {X 0,Y 77.598,Z 285.641,A -85,B 0,C 180,E1 -29893.085,E2 -29893.085} C_VEL
LIN {X 0,Y 76.28,Z 288.417,A -85,B 0,C 180,E1 -29897.894,E2 -29897.894} C_VEL
LIN {X 0,Y 74.854,Z 290.341,A -85,B 0,C 180,E1 -29900.156,E2 -29900.156} C_VEL
LIN {X 0,Y 73.484,Z 291.725,A -85,B 0,C 180,E1 -29901.194,E2 -29901.194} C_VEL
LIN {X 0,Y 65.856,Z 297.778,A -85,B 0,C 180,E1 -29904.918,E2 -29904.918} C_VEL
LIN {X 0,Y 57.179,Z 303.727,A -85,B 0,C 180,E1 -29910.656,E2 -29910.656} C_VEL
LIN {X 0,Y 49.134,Z 308.419,A -85,B 0,C 180,E1 -29918.135,E2 -29918.135} C_VEL
LIN {X 0,Y 42.203,Z 312,A -85,B 0,C 180,E1 -29928.244,E2 -29928.244} C_VEL
LIN {X 0,Y 38.596,Z 313.842,A -85,B 0,C 180,E1 -29936.9,E2 -29936.9} C_VEL
LIN {X 0,Y 35.957,Z 315.224,A -85,B 0,C 180,E1 -29946.999,E2 -29946.999} C_VEL
LIN {X 0,Y 34.465,Z 316.211,A -85,B 0,C 180,E1 -29958.243,E2 -29958.243} C_VEL
LIN {X 0,Y 34.174,Z 316.805,A -85,B 0,C 180,E1 -29970.008,E2 -29970.008} C_VEL
LIN {X 0,Y 34.47,Z 316.973,A -85,B 0,C 180,E1 -29981.772,E2 -29981.772} C_VEL
LIN {X 0,Y 38.644,Z 316.071,A -85,B 0,C 180,E1 -30003.071,E2 -30003.071} C_VEL
LIN {X 0,Y 42.28,Z 315.043,A -85,B 0,C 180,E1 -30011.68,E2 -30011.68} C_VEL
LIN {X 0,Y 46.776,Z 313.609,A -85,B 0,C 180,E1 -30018.702,E2 -30018.702} C_VEL
LIN {X 0,Y 54.488,Z 310.635,A -85,B 0,C 180,E1 -30026.972,E2 -30026.972} C_VEL
LIN {X 0,Y 63.069,Z 306.627,A -85,B 0,C 180,E1 -30033.06,E2 -30033.06} C_VEL
LIN {X 0,Y 73.677,Z 300.472,A -85,B 0,C 180,E1 -30038.44,E2 -30038.44} C_VEL
LIN {X 0,Y 78.402,Z 297.304,A -85,B 0,C 180,E1 -30040.257,E2 -30040.257} C_VEL
LIN {X 0,Y 79.48,Z 296.137,A -85,B 0,C 180,E1 -30041.975,E2 -30041.975} C_VEL
LIN {X 0,Y 80.987,Z 293.868,A -85,B 0,C 180,E1 -30046.551,E2 -30046.551} C_VEL
LIN {X 0,Y 81.741,Z 292.558,A -85,B 0,C 180,E1 -30050.099,E2 -30050.099} C_VEL
LIN {X 0,Y 82.435,Z 291.265,A -85,B 0,C 180,E1 -30055.11,E2 -30055.11} C_VEL
LIN {X 0,Y 82.899,Z 290.572,A -85,B 0,C 180,E1 -30060.001,E2 -30060.001} C_VEL
LIN {X 0,Y 81.822,Z 291.718,A -85,B 0,C 180,E1 -30067.333,E2 -30067.333} C_VEL
LIN {X 0,Y 81.594,Z 292.216,A -85,B 0,C 180,E1 -30069.921,E2 -30069.921} C_VEL
LIN {X 0,Y 80.966,Z 293.648,A -85,B 0,C 180,E1 -30075.095,E2 -30075.095} C_VEL
LIN {X 0,Y 79.809,Z 295.298,A -85,B 0,C 180,E1 -30078.801,E2 -30078.801} C_VEL
LIN {X 0,Y 72.028,Z 300.451,A -85,B 0,C 180,E1 -30082.036,E2 -30082.036} C_VEL
LIN {X 0,Y 63.034,Z 305.434,A -85,B 0,C 180,E1 -30086.878,E2 -30086.878} C_VEL
LIN {X 0,Y 54.616,Z 309.286,A -85,B 0,C 180,E1 -30093.233,E2 -30093.233} C_VEL
LIN {X 0,Y 46.932,Z 312.116,A -85,B 0,C 180,E1 -30101.515,E2 -30101.515} C_VEL
LIN {X 0,Y 38.954,Z 314.383,A -85,B 0,C 180,E1 -30117.226,E2 -30117.226} C_VEL
LIN {X 0,Y 36.246,Z 314.938,A -85,B 0,C 180,E1 -30127.177,E2 -30127.177} C_VEL
LIN {X 0,Y 34.657,Z 315.081,A -85,B 0,C 180,E1 -30138.293,E2 -30138.293} C_VEL
LIN {X 0,Y 34.311,Z 314.818,A -85,B 0,C 180,E1 -30149.992,E2 -30149.992} C_VEL
LIN {X 0,Y 35.152,Z 314.179,A -85,B 0,C 180,E1 -30161.524,E2 -30161.524} C_VEL
LIN {X 0,Y 37.038,Z 313.164,A -85,B 0,C 180,E1 -30172.293,E2 -30172.293} C_VEL
LIN {X 0,Y 39.996,Z 311.728,A -85,B 0,C 180,E1 -30181.803,E2 -30181.803} C_VEL
LIN {X 0,Y 45.986,Z 308.781,A -85,B 0,C 180,E1 -30193.439,E2 -30193.439} C_VEL
LIN {X 0,Y 53.355,Z 304.794,A -85,B 0,C 180,E1 -30202.202,E2 -30202.202} C_VEL
LIN {X 0,Y 63.093,Z 298.65,A -85,B 0,C 180,E1 -30209.671,E2 -30209.671} C_VEL
LIN {X 0,Y 72.043,Z 291.957,A -85,B 0,C 180,E1 -30214.453,E2 -30214.453} C_VEL
LIN {X 0,Y 75.849,Z 288.712,A -85,B 0,C 180,E1 -30216.167,E2 -30216.167} C_VEL
LIN {X 0,Y 76.3,Z 288.066,A -85,B 0,C 180,E1 -30217.068,E2 -30217.068} C_VEL
LIN {X 0,Y 76.758,Z 286.709,A -85,B 0,C 180,E1 -30219.993,E2 -30219.993} C_VEL
LIN {X 0,Y 77.233,Z 285.093,A -85,B 0,C 180,E1 -30224.156,E2 -30224.156} C_VEL
LIN {X 0,Y 77.656,Z 283.355,A -85,B 0,C 180,E1 -30231.094,E2 -30231.094} C_VEL
LIN {X 0,Y 78.008,Z 282.675,A -85,B 0,C 180,E1 -30234.83,E2 -30234.83} C_VEL
LIN {X 0,Y 78.567,Z 282.17,A -85,B 0,C 180,E1 -30239.999,E2 -30239.999} C_VEL
LIN {X 0,Y 78.126,Z 283.13,A -85,B 0,C 180,E1 -30244.879,E2 -30244.879} C_VEL
LIN {X 0,Y 77.536,Z 284.25,A -85,B 0,C 180,E1 -30247.776,E2 -30247.776} C_VEL
LIN {X 0,Y 76.194,Z 286.037,A -85,B 0,C 180,E1 -30250.409,E2 -30250.409} C_VEL
LIN {X 0,Y 73.557,Z 289.022,A -85,B 0,C 180,E1 -30253.495,E2 -30253.495} C_VEL
LIN {X 0,Y 70.106,Z 292.292,A -85,B 0,C 180,E1 -30256.027,E2 -30256.027} C_VEL
LIN {X 0,Y 68.08,Z 293.907,A -85,B 0,C 180,E1 -30256.984,E2 -30256.984} C_VEL
LIN {X 0,Y 58.053,Z 300.914,A -85,B 0,C 180,E1 -30261.542,E2 -30261.542} C_VEL
LIN {X 0,Y 47.918,Z 306.735,A -85,B 0,C 180,E1 -30268.376,E2 -30268.376} C_VEL
LIN {X 0,Y 39.683,Z 310.691,A -85,B 0,C 180,E1 -30277.176,E2 -30277.176} C_VEL
LIN {X 0,Y 32.846,Z 313.617,A -85,B 0,C 180,E1 -30290.08,E2 -30290.08} C_VEL
LIN {X 0,Y 29.518,Z 315.006,A -85,B 0,C 180,E1 -30301.576,E2 -30301.576} C_VEL
LIN {X 0,Y 27.534,Z 315.999,A -85,B 0,C 180,E1 -30315.223,E2 -30315.223} C_VEL
LIN {X 0,Y 27.066,Z 316.599,A -85,B 0,C 180,E1 -30330.01,E2 -30330.01} C_VEL
LIN {X 0,Y 27.54,Z 316.777,A -85,B 0,C 180,E1 -30344.794,E2 -30344.794} C_VEL
LIN {X 0,Y 32.907,Z 315.887,A -85,B 0,C 180,E1 -30369.853,E2 -30369.853} C_VEL
LIN {X 0,Y 37.254,Z 314.863,A -85,B 0,C 180,E1 -30378.997,E2 -30378.997} C_VEL
LIN {X 0,Y 42.406,Z 313.439,A -85,B 0,C 180,E1 -30385.967,E2 -30385.967} C_VEL
LIN {X 0,Y 50.956,Z 310.475,A -85,B 0,C 180,E1 -30393.704,E2 -30393.704} C_VEL
LIN {X 0,Y 60.17,Z 306.479,A -85,B 0,C 180,E1 -30399.137,E2 -30399.137} C_VEL
LIN {X 0,Y 71.372,Z 300.342,A -85,B 0,C 180,E1 -30403.756,E2 -30403.756} C_VEL
LIN {X 0,Y 73.009,Z 299.331,A -85,B 0,C 180,E1 -30404.284,E2 -30404.284} C_VEL
LIN {X 0,Y 74.737,Z 297.772,A -85,B 0,C 180,E1 -30406.919,E2 -30406.919} C_VEL
LIN {X 0,Y 75.375,Z 296.926,A -85,B 0,C 180,E1 -30409.254,E2 -30409.254} C_VEL
LIN {X 0,Y 76.404,Z 295.517,A -85,B 0,C 180,E1 -30414.723,E2 -30414.723} C_VEL
LIN {X 0,Y 77.053,Z 294.764,A -85,B 0,C 180,E1 -30420.001,E2 -30420.001} C_VEL
LIN {X 0,Y 75.908,Z 295.692,A -85,B 0,C 180,E1 -30426.787,E2 -30426.787} C_VEL
LIN {X 0,Y 75.106,Z 296.934,A -85,B 0,C 180,E1 -30432.891,E2 -30432.891} C_VEL
LIN {X 0,Y 74.387,Z 297.723,A -85,B 0,C 180,E1 -30435.001,E2 -30435.001} C_VEL
LIN {X 0,Y 63.266,Z 304.037,A -85,B 0,C 180,E1 -30439.225,E2 -30439.225} C_VEL
LIN {X 0,Y 54.011,Z 308.266,A -85,B 0,C 180,E1 -30444.374,E2 -30444.374} C_VEL
LIN {X 0,Y 48.146,Z 310.504,A -85,B 0,C 180,E1 -30448.852,E2 -30448.852} C_VEL
LIN {X 0,Y 42.547,Z 312.29,A -85,B 0,C 180,E1 -30454.315,E2 -30454.315} C_VEL
LIN {X 0,Y 33.19,Z 314.568,A -85,B 0,C 180,E1 -30470.554,E2 -30470.554} C_VEL
LIN {X 0,Y 29.83,Z 315.128,A -85,B 0,C 180,E1 -30481.879,E2 -30481.879} C_VEL
LIN {X 0,Y 27.73,Z 315.282,A -85,B 0,C 180,E1 -30495.31,E2 -30495.31} C_VEL
LIN {X 0,Y 27.228,Z 315.023,A -85,B 0,C 180,E1 -30509.99,E2 -30509.99} C_VEL
LIN {X 0,Y 28.251,Z 314.39,A -85,B 0,C 180,E1 -30524.394,E2 -30524.394} C_VEL
LIN {X 0,Y 30.598,Z 313.381,A -85,B 0,C 180,E1 -30537.335,E2 -30537.335} C_VEL
LIN {X 0,Y 34.171,Z 311.957,A -85,B 0,C 180,E1 -30548.085,E2 -30548.085} C_VEL
LIN {X 0,Y 41.132,Z 309.02,A -85,B 0,C 180,E1 -30560.239,E2 -30560.239} C_VEL
LIN {X 0,Y 49.336,Z 305.044,A -85,B 0,C 180,E1 -30568.71,E2 -30568.71} C_VEL
LIN {X 0,Y 59.83,Z 298.917,A -85,B 0,C 180,E1 -30575.535,E2 -30575.535} C_VEL
LIN {X 0,Y 69.082,Z 292.394,A -85,B 0,C 180,E1 -30579.666,E2 -30579.666} C_VEL
LIN {X 0,Y 70.473,Z 291.326,A -85,B 0,C 180,E1 -30580.212,E2 -30580.212} C_VEL
LIN {X 0,Y 71.254,Z 290.121,A -85,B 0,C 180,E1 -30582.787,E2 -30582.787} C_VEL
LIN {X 0,Y 71.945,Z 288.488,A -85,B 0,C 180,E1 -30588.732,E2 -30588.732} C_VEL
LIN {X 0,Y 72.56,Z 287.445,A -85,B 0,C 180,E1 -30594.44,E2 -30594.44} C_VEL
LIN {X 0,Y 73.164,Z 286.944,A -85,B 0,C 180,E1 -30599.999,E2 -30599.999} C_VEL
LIN {X 0,Y 72.662,Z 287.952,A -85,B 0,C 180,E1 -30605.549,E2 -30605.549} C_VEL
LIN {X 0,Y 72.106,Z 289.513,A -85,B 0,C 180,E1 -30611.24,E2 -30611.24} C_VEL
LIN {X 0,Y 71.168,Z 291.009,A -85,B 0,C 180,E1 -30614.289,E2 -30614.289} C_VEL
LIN {X 0,Y 69.593,Z 292.746,A -85,B 0,C 180,E1 -30616.414,E2 -30616.414} C_VEL
LIN {X 0,Y 68.08,Z 293.907,A -85,B 0,C 180,E1 -30616.984,E2 -30616.984} C_VEL
LIN {X 0,Y 63.384,Z 297.2,A -85,B 0,C 180,E1 -30618.273,E2 -30618.273} C_VEL
LIN {X 0,Y 54.785,Z 302.041,A -85,B 0,C 180,E1 -30619.269,E2 -30619.269} C_VEL
LIN {X 0,Y 45.859,Z 306.21,A -85,B 0,C 180,E1 -30620.773,E2 -30620.773} C_VEL
LIN {X 0,Y 40.746,Z 308.397,A -85,B 0,C 180,E1 -30623.462,E2 -30623.462} C_VEL
LIN {X 0,Y 32.955,Z 311.53,A -85,B 0,C 180,E1 -30631.48,E2 -30631.48} C_VEL
LIN {X 0,Y 27.755,Z 313.392,A -85,B 0,C 180,E1 -30640.587,E2 -30640.587} C_VEL
LIN {X 0,Y 23.495,Z 314.788,A -85,B 0,C 180,E1 -30653.273,E2 -30653.273} C_VEL
LIN {X 0,Y 20.741,Z 315.787,A -85,B 0,C 180,E1 -30670.208,E2 -30670.208} C_VEL
LIN {X 0,Y 19.971,Z 316.393,A -85,B 0,C 180,E1 -30690.014,E2 -30690.014} C_VEL
LIN {X 0,Y 20.748,Z 316.58,A -85,B 0,C 180,E1 -30709.812,E2 -30709.812} C_VEL
LIN {X 0,Y 27.807,Z 315.702,A -85,B 0,C 180,E1 -30739.318,E2 -30739.318} C_VEL
LIN {X 0,Y 33.015,Z 314.684,A -85,B 0,C 180,E1 -30748.384,E2 -30748.384} C_VEL
LIN {X 0,Y 38.865,Z 313.269,A -85,B 0,C 180,E1 -30754.716,E2 -30754.716} C_VEL
LIN {X 0,Y 48.227,Z 310.315,A -85,B 0,C 180,E1 -30761.308,E2 -30761.308} C_VEL
LIN {X 0,Y 59.781,Z 305.486,A -85,B 0,C 180,E1 -30766.402,E2 -30766.402} C_VEL
LIN {X 0,Y 67.73,Z 301.372,A -85,B 0,C 180,E1 -30768.892,E2 -30768.892} C_VEL
LIN {X 0,Y 70.024,Z 299.449,A -85,B 0,C 180,E1 -30774.241,E2 -30774.241} C_VEL
LIN {X 0,Y 70.435,Z 299.057,A -85,B 0,C 180,E1 -30776.199,E2 -30776.199} C_VEL
LIN {X 0,Y 70.934,Z 298.597,A -85,B 0,C 180,E1 -30780.001,E2 -30780.001} C_VEL
LIN {X 0,Y 69.507,Z 299.645,A -85,B 0,C 180,E1 -30788.213,E2 -30788.213} C_VEL
LIN {X 0,Y 69.359,Z 299.834,A -85,B 0,C 180,E1 -30789.443,E2 -30789.443} C_VEL
LIN {X 0,Y 67.637,Z 300.905,A -85,B 0,C 180,E1 -30790.934,E2 -30790.934} C_VEL
LIN {X 0,Y 57.994,Z 305.732,A -85,B 0,C 180,E1 -30794.189,E2 -30794.189} C_VEL
LIN {X 0,Y 48.291,Z 309.609,A -85,B 0,C 180,E1 -30798.916,E2 -30798.916} C_VEL
LIN {X 0,Y 38.981,Z 312.463,A -85,B 0,C 180,E1 -30805.642,E2 -30805.642} C_VEL
LIN {X 0,Y 28.046,Z 314.753,A -85,B 0,C 180,E1 -30821.246,E2 -30821.246} C_VEL
LIN {X 0,Y 23.783,Z 315.318,A -85,B 0,C 180,E1 -30833.761,E2 -30833.761} C_VEL
LIN {X 0,Y 20.941,Z 315.482,A -85,B 0,C 180,E1 -30850.378,E2 -30850.378} C_VEL
LIN {X 0,Y 20.119,Z 315.23,A -85,B 0,C 180,E1 -30869.986,E2 -30869.986} C_VEL
LIN {X 0,Y 21.451,Z 314.602,A -85,B 0,C 180,E1 -30889.11,E2 -30889.11} C_VEL
LIN {X 0,Y 24.508,Z 313.598,A -85,B 0,C 180,E1 -30904.98,E2 -30904.98} C_VEL
LIN {X 0,Y 28.914,Z 312.185,A -85,B 0,C 180,E1 -30916.8,E2 -30916.8} C_VEL
LIN {X 0,Y 37.008,Z 309.257,A -85,B 0,C 180,E1 -30928.692,E2 -30928.692} C_VEL
LIN {X 0,Y 46.053,Z 305.295,A -85,B 0,C 180,E1 -30936.272,E2 -30936.272} C_VEL
LIN {X 0,Y 57.252,Z 299.185,A -85,B 0,C 180,E1 -30942.026,E2 -30942.026} C_VEL
LIN {X 0,Y 65.476,Z 293.749,A -85,B 0,C 180,E1 -30944.991,E2 -30944.991} C_VEL
LIN {X 0,Y 65.917,Z 293.055,A -85,B 0,C 180,E1 -30947.686,E2 -30947.686} C_VEL
LIN {X 0,Y 66.771,Z 291.936,A -85,B 0,C 180,E1 -30953.957,E2 -30953.957} C_VEL
LIN {X 0,Y 67.516,Z 291.407,A -85,B 0,C 180,E1 -30959.999,E2 -30959.999} C_VEL
LIN {X 0,Y 66.798,Z 292.475,A -85,B 0,C 180,E1 -30966.038,E2 -30966.038} C_VEL
LIN {X 0,Y 66.462,Z 293.1,A -85,B 0,C 180,E1 -30968.663,E2 -30968.663} C_VEL
LIN {X 0,Y 64.564,Z 294.941,A -85,B 0,C 180,E1 -30971.612,E2 -30971.612} C_VEL
LIN {X 0,Y 54.927,Z 301.196,A -85,B 0,C 180,E1 -30975.078,E2 -30975.078} C_VEL
LIN {X 0,Y 44.966,Z 306.488,A -85,B 0,C 180,E1 -30980.349,E2 -30980.349} C_VEL
LIN {X 0,Y 40.746,Z 308.397,A -85,B 0,C 180,E1 -30983.462,E2 -30983.462} C_VEL
LIN {X 0,Y 35.689,Z 310.38,A -85,B 0,C 180,E1 -30987,E2 -30987} C_VEL
LIN {X 0,Y 26.672,Z 313.014,A -85,B 0,C 180,E1 -30992.802,E2 -30992.802} C_VEL
LIN {X 0,Y 19.594,Z 314.578,A -85,B 0,C 180,E1 -31001.002,E2 -31001.002} C_VEL
LIN {X 0,Y 15.234,Z 315.387,A -85,B 0,C 180,E1 -31014.071,E2 -31014.071} C_VEL
LIN {X 0,Y 14.223,Z 315.579,A -85,B 0,C 180,E1 -31020.638,E2 -31020.638} C_VEL
LIN {X 0,Y 12.867,Z 316.187,A -85,B 0,C 180,E1 -31050.021,E2 -31050.021} C_VEL
LIN {X 0,Y 14.253,Z 316.382,A -85,B 0,C 180,E1 -31079.563,E2 -31079.563} C_VEL
LIN {X 0,Y 23.783,Z 315.517,A -85,B 0,C 180,E1 -31112.453,E2 -31112.453} C_VEL
LIN {X 0,Y 29.9,Z 314.504,A -85,B 0,C 180,E1 -31120.103,E2 -31120.103} C_VEL
LIN {X 0,Y 36.396,Z 313.098,A -85,B 0,C 180,E1 -31124.917,E2 -31124.917} C_VEL
LIN {X 0,Y 46.439,Z 310.154,A -85,B 0,C 180,E1 -31129.65,E2 -31129.65} C_VEL
LIN {X 0,Y 57.556,Z 305.794,A -85,B 0,C 180,E1 -31132.988,E2 -31132.988} C_VEL
LIN {X 0,Y 60.111,Z 304.59,A -85,B 0,C 180,E1 -31133.584,E2 -31133.584} C_VEL
LIN {X 0,Y 63.473,Z 302.876,A -85,B 0,C 180,E1 -31135.214,E2 -31135.214} C_VEL
LIN {X 0,Y 64.622,Z 302.07,A -85,B 0,C 180,E1 -31140.001,E2 -31140.001} C_VEL
LIN {X 0,Y 63.549,Z 302.658,A -85,B 0,C 180,E1 -31145.542,E2 -31145.542} C_VEL
LIN {X 0,Y 53.255,Z 307.296,A -85,B 0,C 180,E1 -31148.196,E2 -31148.196} C_VEL
LIN {X 0,Y 43.118,Z 310.827,A -85,B 0,C 180,E1 -31152.037,E2 -31152.037} C_VEL
LIN {X 0,Y 36.472,Z 312.635,A -85,B 0,C 180,E1 -31155.517,E2 -31155.517} C_VEL
LIN {X 0,Y 23.951,Z 314.937,A -85,B 0,C 180,E1 -31168.304,E2 -31168.304} C_VEL
LIN {X 0,Y 18.528,Z 315.508,A -85,B 0,C 180,E1 -31180.637,E2 -31180.637} C_VEL
LIN {X 0,Y 14.46,Z 315.682,A -85,B 0,C 180,E1 -31200.9,E2 -31200.9} C_VEL
LIN {X 0,Y 13.013,Z 315.436,A -85,B 0,C 180,E1 -31229.979,E2 -31229.979} C_VEL
LIN {X 0,Y 14.942,Z 314.813,A -85,B 0,C 180,E1 -31258.035,E2 -31258.035} C_VEL
LIN {X 0,Y 19.133,Z 313.816,A -85,B 0,C 180,E1 -31277.253,E2 -31277.253} C_VEL
LIN {X 0,Y 24.609,Z 312.413,A -85,B 0,C 180,E1 -31288.926,E2 -31288.926} C_VEL
LIN {X 0,Y 33.865,Z 309.495,A -85,B 0,C 180,E1 -31299.014,E2 -31299.014} C_VEL
LIN {X 0,Y 43.681,Z 305.544,A -85,B 0,C 180,E1 -31304.835,E2 -31304.835} C_VEL
LIN {X 0,Y 53.786,Z 300.448,A -85,B 0,C 180,E1 -31308.477,E2 -31308.477} C_VEL
LIN {X 0,Y 59.679,Z 296.906,A -85,B 0,C 180,E1 -31310.062,E2 -31310.062} C_VEL
LIN {X 0,Y 60.641,Z 296.114,A -85,B 0,C 180,E1 -31313.343,E2 -31313.343} C_VEL
LIN {X 0,Y 61.561,Z 295.542,A -85,B 0,C 180,E1 -31319.998,E2 -31319.998} C_VEL
LIN {X 0,Y 61.097,Z 296.027,A -85,B 0,C 180,E1 -31323.181,E2 -31323.181} C_VEL
LIN {X 0,Y 59.912,Z 297.044,A -85,B 0,C 180,E1 -31326.053,E2 -31326.053} C_VEL
LIN {X 0,Y 49.791,Z 302.943,A -85,B 0,C 180,E1 -31328.928,E2 -31328.928} C_VEL
LIN {X 0,Y 39.667,Z 307.677,A -85,B 0,C 180,E1 -31333.025,E2 -31333.025} C_VEL
LIN {X 0,Y 29.859,Z 311.295,A -85,B 0,C 180,E1 -31339.736,E2 -31339.736} C_VEL
LIN {X 0,Y 23.732,Z 313.165,A -85,B 0,C 180,E1 -31347.359,E2 -31347.359} C_VEL
LIN {X 0,Y 18.292,Z 314.571,A -85,B 0,C 180,E1 -31359.815,E2 -31359.815} C_VEL
LIN {X 0,Y 14.223,Z 315.579,A -85,B 0,C 180,E1 -31380.638,E2 -31380.638} C_VEL
LIN {X 0,Y 12.629,Z 315.961,A -85,B 0,C 180,E1 -31395.976,E2 -31395.976} C_VEL
LIN {X 0,Y 11.481,Z 316.199,A -85,B 0,C 180,E1 -31413.954,E2 -31413.954} C_VEL
LIN {X 0,Y 11.998,Z 316.257,A -85,B 0,C 180,E1 -31453.521,E2 -31453.521} C_VEL
LIN {X 0,Y 16.67,Z 315.883,A -85,B 0,C 180,E1 -31480.455,E2 -31480.455} C_VEL
LIN {X 0,Y 21.803,Z 315.291,A -85,B 0,C 180,E1 -31489.715,E2 -31489.715} C_VEL
LIN {X 0,Y 23.689,Z 314.998,A -85,B 0,C 180,E1 -31491.293,E2 -31491.293} C_VEL
LIN {X 0,Y 35.22,Z 312.927,A -85,B 0,C 180,E1 -31496.182,E2 -31496.182} C_VEL
LIN {X 0,Y 45.7,Z 309.992,A -85,B 0,C 180,E1 -31498.454,E2 -31498.454} C_VEL
LIN {X 0,Y 55.913,Z 306.156,A -85,B 0,C 180,E1 -31500.002,E2 -31500.002} C_VEL
LIN {X 0,Y 45.703,Z 309.933,A -85,B 0,C 180,E1 -31501.697,E2 -31501.697} C_VEL
LIN {X 0,Y 35.242,Z 312.807,A -85,B 0,C 180,E1 -31504.311,E2 -31504.311} C_VEL
LIN {X 0,Y 21.507,Z 315.122,A -85,B 0,C 180,E1 -31511.343,E2 -31511.343} C_VEL
LIN {X 0,Y 14.908,Z 315.698,A -85,B 0,C 180,E1 -31519.424,E2 -31519.424} C_VEL
LIN {X 0,Y 8.943,Z 315.881,A -85,B 0,C 180,E1 -31538.157,E2 -31538.157} C_VEL
LIN {X 0,Y 5.922,Z 315.642,A -85,B 0,C 180,E1 -31589.954,E2 -31589.954} C_VEL
LIN {X 0,Y 9.303,Z 315.024,A -85,B 0,C 180,E1 -31639.016,E2 -31639.016} C_VEL
LIN {X 0,Y 15.24,Z 314.032,A -85,B 0,C 180,E1 -31657.207,E2 -31657.207} C_VEL
LIN {X 0,Y 21.814,Z 312.64,A -85,B 0,C 180,E1 -31665.069,E2 -31665.069} C_VEL
LIN {X 0,Y 32.018,Z 309.732,A -85,B 0,C 180,E1 -31670.949,E2 -31670.949} C_VEL
LIN {X 0,Y 42.381,Z 305.794,A -85,B 0,C 180,E1 -31674.146,E2 -31674.146} C_VEL
LIN {X 0,Y 53.87,Z 300.121,A -85,B 0,C 180,E1 -31676.215,E2 -31676.215} C_VEL
LIN {X 0,Y 55.051,Z 299.459,A -85,B 0,C 180,E1 -31678.049,E2 -31678.049} C_VEL
LIN {X 0,Y 53.31,Z 300.508,A -85,B 0,C 180,E1 -31679.998,E2 -31679.998} C_VEL
LIN {X 0,Y 42.183,Z 305.993,A -85,B 0,C 180,E1 -31681.88,E2 -31681.88} C_VEL
LIN {X 0,Y 31.727,Z 309.986,A -85,B 0,C 180,E1 -31684.737,E2 -31684.737} C_VEL
LIN {X 0,Y 21.41,Z 312.938,A -85,B 0,C 180,E1 -31690.112,E2 -31690.112} C_VEL
LIN {X 0,Y 14.778,Z 314.353,A -85,B 0,C 180,E1 -31698.061,E2 -31698.061} C_VEL
LIN {X 0,Y 8.385,Z 315.411,A -85,B 0,C 180,E1 -31719.363,E2 -31719.363} C_VEL
LIN {X 0,Y 5.754,Z 315.981,A -85,B 0,C 180,E1 -31770.047,E2 -31770.047} C_VEL
LIN {X 0,Y 8.798,Z 316.184,A -85,B 0,C 180,E1 -31823.06,E2 -31823.06} C_VEL
LIN {X 0,Y 14.802,Z 315.953,A -85,B 0,C 180,E1 -31841.781,E2 -31841.781} C_VEL
LIN {X 0,Y 23.689,Z 314.998,A -85,B 0,C 180,E1 -31851.293,E2 -31851.293} C_VEL
LIN {X 0,Y 25.898,Z 316.978,A -85,B 0,C 180,E1 -31852.618,E2 -31852.618} C_VEL
LIN {X 0,Y 25.898,Z 600,A -85,B 0,C 180,E1 -31852.618,E2 -31852.618} C_VEL
LIN {X 0,Y 25.898,Z 600,A -85,B 0,C 180,E1 -31852.618,E2 -31852.618}

QRS_NEXT_CUT()

QRS_NEXT()
QRS_HOME()

END
